(* PLC project Unnamed, Unknown Unnamed 1 *)
(* stored: creationDateTime 2020-09-16T10:44:23, modificationDateTime 2020-09-16T18:36:56 *)

PROGRAM SimpleProgram1
  VAR
    s1 : BOOL := FALSE;
    MOTOR : BOOL;
  END_VAR

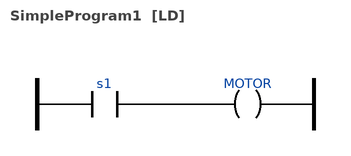
(* LD diagram, written out as Structured Text *)
MOTOR := s1;
END_PROGRAM

CONFIGURATION Config0
  RESOURCE Res0 ON PLC
    TASK task0(INTERVAL := T#20ms, PRIORITY := 0);
    PROGRAM instance0 WITH task0 : SimpleProgram1;
  END_RESOURCE
END_CONFIGURATION
